Universal Robots PolyScope program: U.urp

Program U (installation=default directory=/programs/usbdisk/UR10_Code createdIn=3.15.4.106291 lastSavedIn=3.15.4.106291 robotSerialNumber=2019300133)
Calibrated DH parameters: a=[-0.000006, -0.606471, -0.570201, -0.000053, 0.000006, 0]; d=[0.128096, 15.114888, -22.674746, 7.723348, 0.115665, 0.092162]; alpha=[1.570605, -0.005579, -0.004649, 1.571049, -1.571015, 0]; deltaTheta=[-0.00004, -0.169247, 0.199673, -0.061563, -0.000077, -0.000043]
InitVariablesNode
Robot Program (runOnlyOnce=false)
  SuppressedNode
    Encoder_Target := 0
  SuppressedNode
    Loop While (checkContinuously=false) expression=digital_in[3] ==  True
      CallSubProgram
      Call Orin_Variables
      CallSubProgram
      CallSubProgram
  If digital_out[3] ==  True
    Call Orin_Variables
SubProgram -> Orin_Variables
Thread Thread_1 (runOnlyOnce=false)
  Script: socket_open("192.168.0.3", 50001, "Orin_Encoder")
  Loop Forever
    Encoder_Count := encoder_get_tick_count(0)
    Script: socket_send_line(Encoder_Count, "Orin_Encoder")
    Wait Sleep waitTime=1
SuppressedNode
  Thread Thread_2 (runOnlyOnce=false)
    Script: socket_open("192.168.0.3", 30002, "Boolean")
    Loop Forever
      message := socket_read_string("Boolean")
      If message == "True" (checkContinuously=true)
        ready := True
        var_1 := digital_out[1]== True
      Wait NoWait
SubProgram Orin_Variables (keepSynchronizedWithDisk=false)
  Script: socket_open("192.168.0.3", 50000, "Orin_Target")
  Encoder_Target := socket_get_var("Target_Encoder", "Orin_Target")
  Wait Sleep waitTime=1
  SuppressedNode
    Y := -0.15
